PROGRAM Speed_Setpoints
VAR

	oSpicePumpSpeed: REAL;

	oCloserSpeed: REAL;
	Spare1Setpoint: INT;
	Spare2Setpoint: INT;

	Sp1: INT;
	Sp2: INT;

	Exit_Conv_Speed_SPt: INT;
	test: REAL;
	Spiral_Infeed_Spt: INT;
	Spiral_Infeed_Setpoint: INT;

END_VAR
VAR // added by the converter: edge detectors and wires of the graphical bodies
    _w1, _w2 : ANY;
END_VAR

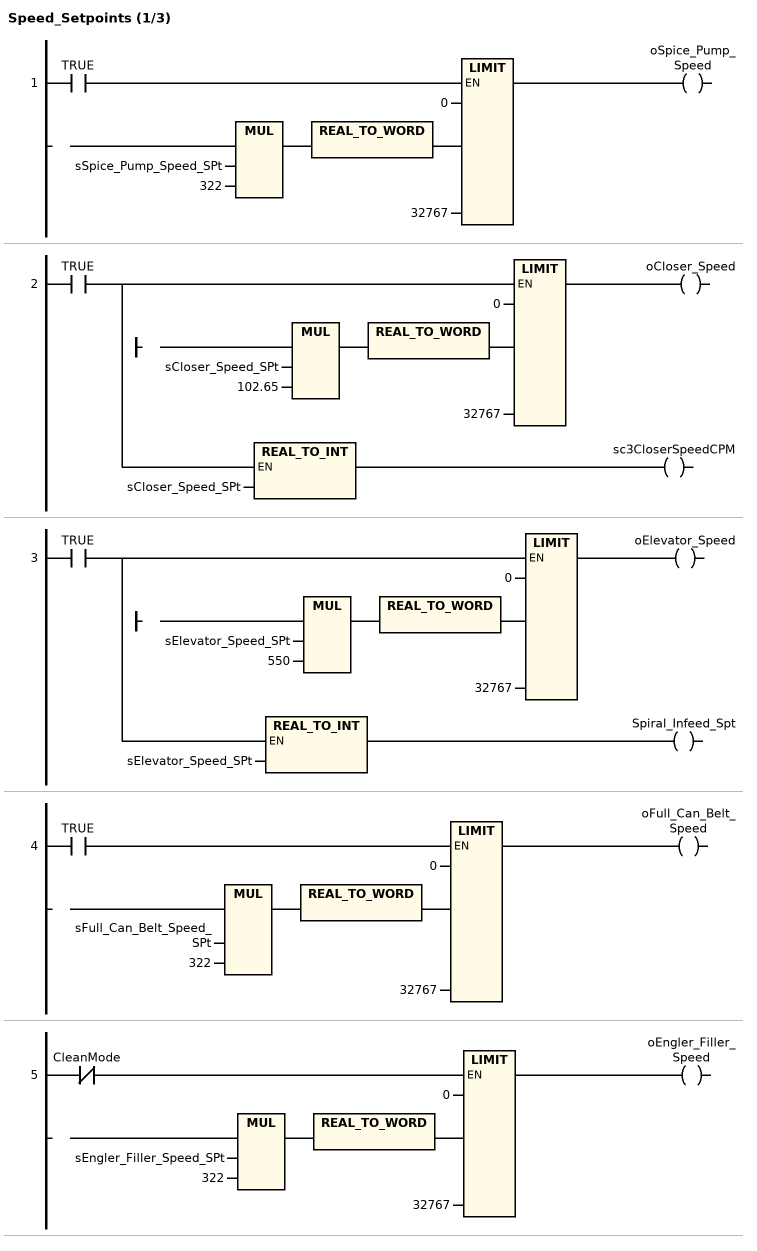
// NETWORK 1
oSpice_Pump_Speed := LIMIT(0, REAL_TO_WORD(sSpice_Pump_Speed_SPt * 322), 32767);

// NETWORK 2
oCloser_Speed := LIMIT(0, REAL_TO_WORD(sCloser_Speed_SPt * 102.65), 32767);
sc3CloserSpeedCPM := REAL_TO_INT(sCloser_Speed_SPt);

// NETWORK 3
oElevator_Speed := LIMIT(0, REAL_TO_WORD(sElevator_Speed_SPt * 550), 32767);
Spiral_Infeed_Spt := REAL_TO_INT(sElevator_Speed_SPt);

// NETWORK 4
oFull_Can_Belt_Speed := LIMIT(0, REAL_TO_WORD(sFull_Can_Belt_Speed_SPt * 322), 32767);

// NETWORK 5
IF NOT CleanMode THEN _w1 := LIMIT(0, REAL_TO_WORD(sEngler_Filler_Speed_SPt * 322), 32767); END_IF
oEngler_Filler_Speed := _w1;

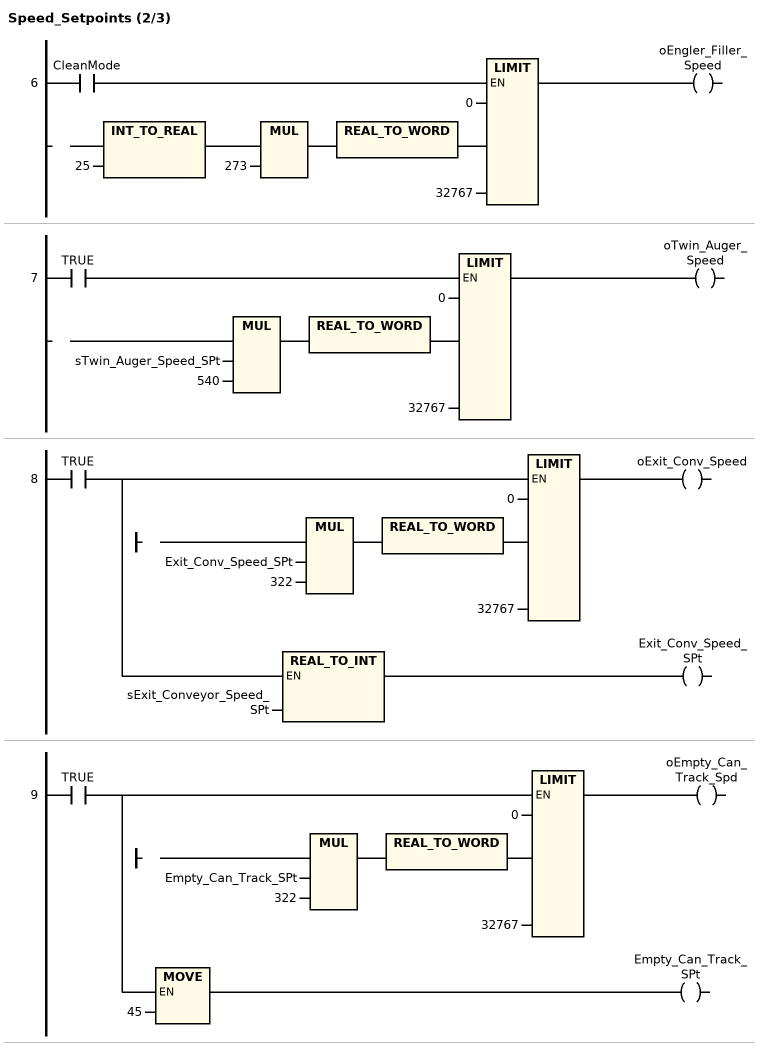
// NETWORK 6
IF CleanMode THEN _w2 := LIMIT(0, REAL_TO_WORD(INT_TO_REAL(25) * 273), 32767); END_IF
oEngler_Filler_Speed := _w2;

// NETWORK 7
oTwin_Auger_Speed := LIMIT(0, REAL_TO_WORD(sTwin_Auger_Speed_SPt * 540), 32767);

// NETWORK 8
oExit_Conv_Speed := LIMIT(0, REAL_TO_WORD(Exit_Conv_Speed_SPt * 322), 32767);
Exit_Conv_Speed_SPt := REAL_TO_INT(sExit_Conveyor_Speed_SPt);

// NETWORK 9
oEmpty_Can_Track_Spd := LIMIT(0, REAL_TO_WORD(Empty_Can_Track_SPt * 322), 32767);
Empty_Can_Track_SPt := 45;

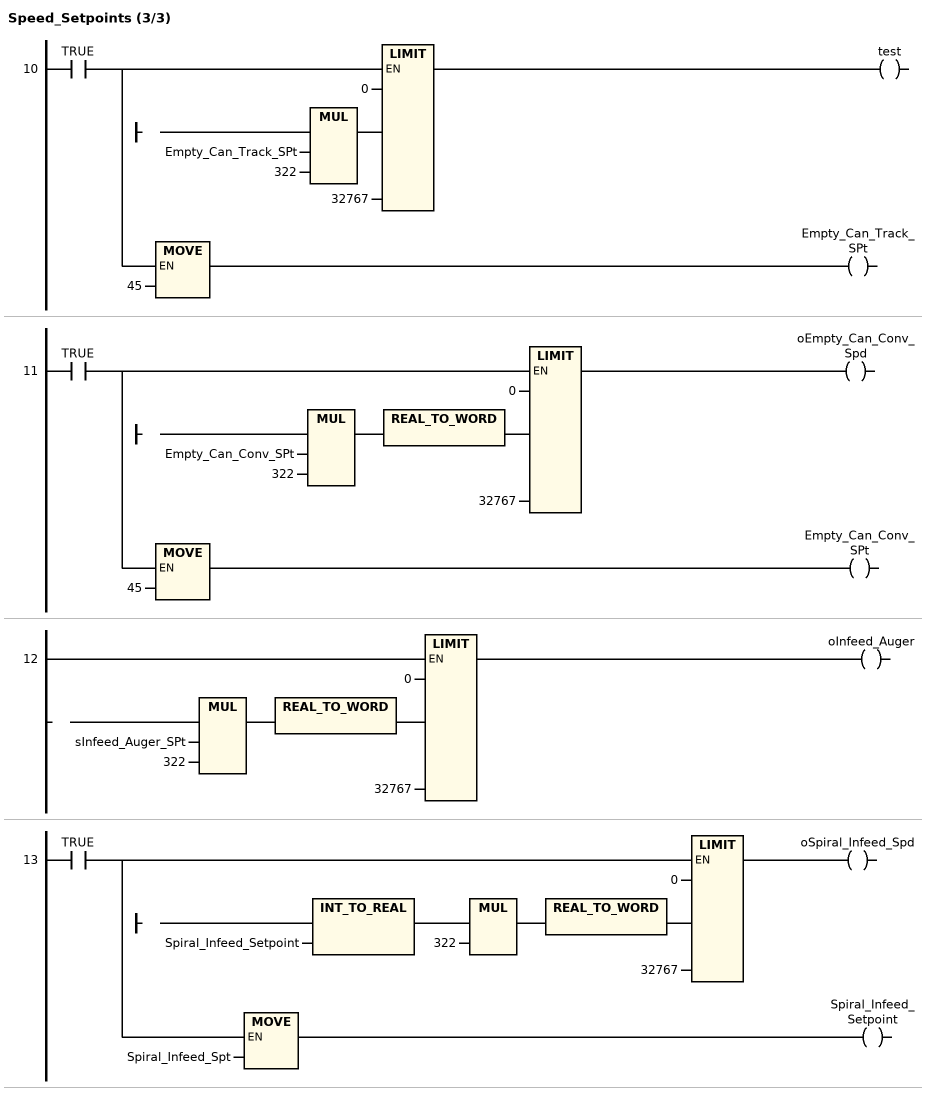
// NETWORK 10
test := LIMIT(0, Empty_Can_Track_SPt * 322, 32767);
Empty_Can_Track_SPt := 45;

// NETWORK 11
oEmpty_Can_Conv_Spd := LIMIT(0, REAL_TO_WORD(Empty_Can_Conv_SPt * 322), 32767);
Empty_Can_Conv_SPt := 45;

// NETWORK 12
oInfeed_Auger := LIMIT(0, REAL_TO_WORD(sInfeed_Auger_SPt * 322), 32767);

// NETWORK 13
oSpiral_Infeed_Spd := LIMIT(0, REAL_TO_WORD(INT_TO_REAL(Spiral_Infeed_Setpoint) * 322), 32767);
Spiral_Infeed_Setpoint := Spiral_Infeed_Spt;

END_PROGRAM

(* stored: Version 1.1.0.1, ProductVersion 3.1.4024.15
   POU Speed_Setpoints: Id {61537346-07b2-493d-ac31-826984faf200}, SpecialFunc None *)
